RoboDK station: New Station 2.0.1..rdk

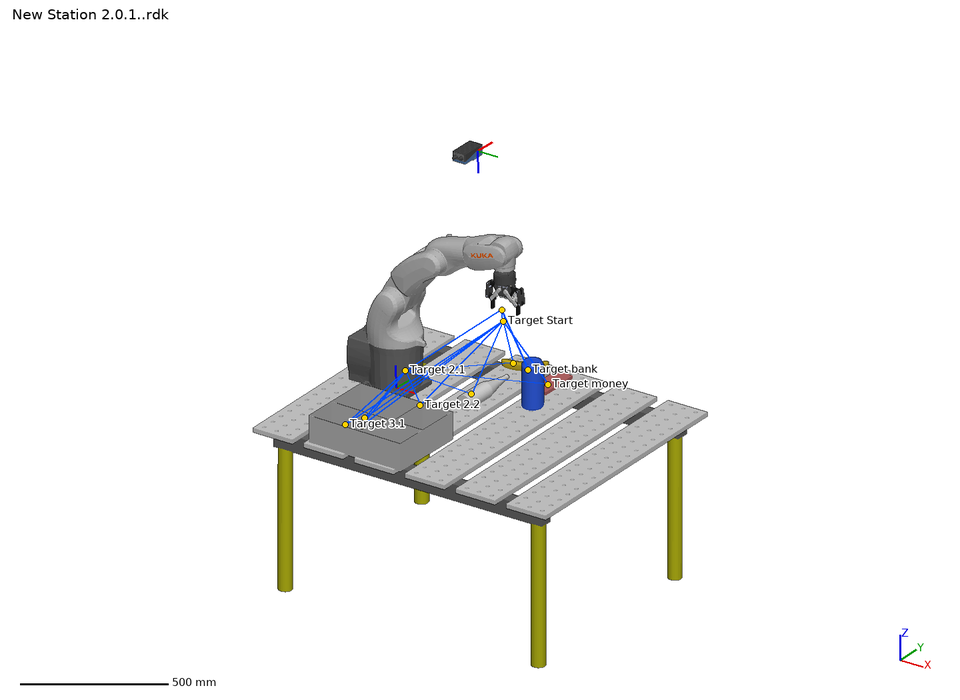
[picture v0: the station drawn from its stored meshes, robots at their saved joint values, targets as dots, program paths as lines]
Station New Station (2). Poses are relative to the parent item; angles as X-Y-Z fixed-axis rotations.
Station parameters (name, value as stored): IO_5, 1, CollisionFreePlanner, KUKA KR 3 R540, CollisionFreePlanner-Rob KUKA KR 3 R540
  - frame KUKA KR 3 R540 Base at (-517.33, 1.06, 0.26) mm, rotated rx -0.44 ry -1.04 rz -0.63 deg
    - robot KUKA KR 3 R540: 6 axes, payload 3 kg, reach 541 mm, repeatability 0.02 mm, weight 26 kg
        modified DH rows (alpha deg, a mm, theta deg, d mm): 0, 0, 0, 345; -90, 20, 0, 0; 0, 260, -90, 0; -90, 20, 0, 260; 90, 0, 0, 0; -90, 0, 180, 75
        joint limits [-170, -170, -110, -175, -120, -350] to [170, 50, 155, 175, 120, 350]; home [0, -90, 90, 0, 0, 0]; saved at [-1.677, -47.408, 34.067, 0.03, 102.342, -1.67]
      - tool Gripper RobotiQ 85 Opened, TCP at (0, -20, 130) mm, size 147.4 x 146.8 x 75 mm
      - tool Gripper RobotiQ 85 Closed, TCP at (0, -20, 130) mm, size 134.4 x 157.6 x 75 mm
    - frame Cam 1 Frame at (362.24, -15.63, 980.06) mm, rotated rx -180 ry -0.87 rz 89.94 deg
      - object Cam 1 at (-36.13, -0.26, 0) mm, rotated rx 0 ry 0 rz -0.06 deg, size 53 x 116 x 38 mm, geometry from Cam2D_SICK_VSPP_5F2113.sld
    - target Target Start (Cartesian target) at (452.7, -7.79, 370.63) mm, rotated rx -180 ry 0 rz 180 deg; joints [-1.545, -47.721, 43.682, 0, 94.039, -1.545] of KUKA KR 3 R540
    - target Target 1 (Cartesian target) at (447.72, -7, 410.9) mm, rotated rx -180 ry 1 rz 180 deg; joints [-1.677, -47.408, 34.067, 0.03, 102.342, -1.67] of KUKA KR 3 R540
    - target Target bank (Cartesian target) at (458.07, 126.15, 139.29) mm, rotated rx 180 ry 0 rz -180 deg; joints [-17.695, -27.719, 59.924, 0, 57.795, -17.695] of KUKA KR 3 R540
    - target Target 2.1 (Cartesian target) at (322.58, -390.29, 298.41) mm, rotated rx 180 ry 1 rz 180 deg; joints [49.256, -36.872, 40.75, -0.76, 85.47, 49.311] of KUKA KR 3 R540
    - target Target 2.2 (Cartesian target) at (321.53, -307.67, 139.3) mm, rotated rx -180 ry 0 rz 180 deg; joints [41.819, -37.777, 80.016, 0, 47.761, 41.819] of KUKA KR 3 R540
    - target Target botlle (Cartesian target) at (290.88, 30.87, 41.6) mm, rotated rx -180 ry 0 rz -180 deg; joints [-9.919, -36.305, 116.095, 0, 10.21, -9.919] of KUKA KR 3 R540
    - target Target 3.1 (Cartesian target) at (123.71, -463.28, 74.82) mm, rotated rx 179 ry 0.04 rz 90 deg; joints [73.166, -17.995, 56.227, -1.21, 51.452, -16.082] of KUKA KR 3 R540
    - target Target banana (Cartesian target) at (247.79, 330.18, 29.97) mm, rotated rx 180 ry 0 rz 120.51 deg; joints [-52.092, -20.233, 74.697, 0, 35.536, -111.581] of KUKA KR 3 R540
    - target Target 3.2 (Cartesian target) at (118.04, -362.03, 29.97) mm, rotated rx 180 ry 0 rz 90.7 deg; joints [69.116, -25.994, 89.591, 0, 26.403, -20.184] of KUKA KR 3 R540
    - target Target money (Cartesian target) at (420.97, 289.96, 12.37) mm, rotated rx -180 ry 0 rz -180 deg; joints [-36.364, 9.152, 14.566, 0, 66.282, -36.364] of KUKA KR 3 R540
    - target Target 3.3 (Cartesian target) at (69.76, -280.26, 13.99) mm, rotated rx 180 ry -0.99 rz 88.58 deg; joints [72.493, -29.84, 112.61, -2.251, 8.17, -16.697] of KUKA KR 3 R540
  - program Prog1 (46 instructions, listed below)
  - program Replace objects (1 instructions, listed below)
  - Python program SimulateToolOpen (listed below)
  - Python program SimulateCamera (listed below)
  - program Target1ToTarget2 (2 instructions, listed below)
  - object  at (-133.86, -215.64, 5.64) mm, rotated rx 90 ry 0 rz -90.4 deg, size 304 x 104 x 379 mm, geometry from  v2.stl
  - object Table at (-140.14, -45.85, 5.02) mm, rotated rx 0 ry 0.02 rz 0.64 deg, size 1193.8 x 965.2 x 609.6 mm, geometry from welding_table.sld
  - object bank v1 at (-54.34, 174.14, 1.34) mm, size 76.9 x 76.9 x 170.3 mm, geometry from bank v1.stl
  - object botlle v1 at (-226.47, -16.86, 5.96) mm, rotated rx -90 ry 0 rz 0 deg, size 60 x 60 x 252.8 mm, geometry from botlle v1.stl
  - object banana v1 at (-288.68, 344.87, 0) mm, rotated rx 0 ry 0 rz -150.16 deg, size 159.5 x 33.3 x 40.6 mm, geometry from banana v1.stl
  - object money v2 at (-132.34, 388.08, 7.15) mm, size 69 x 157 x 12 mm, geometry from money v2.stl
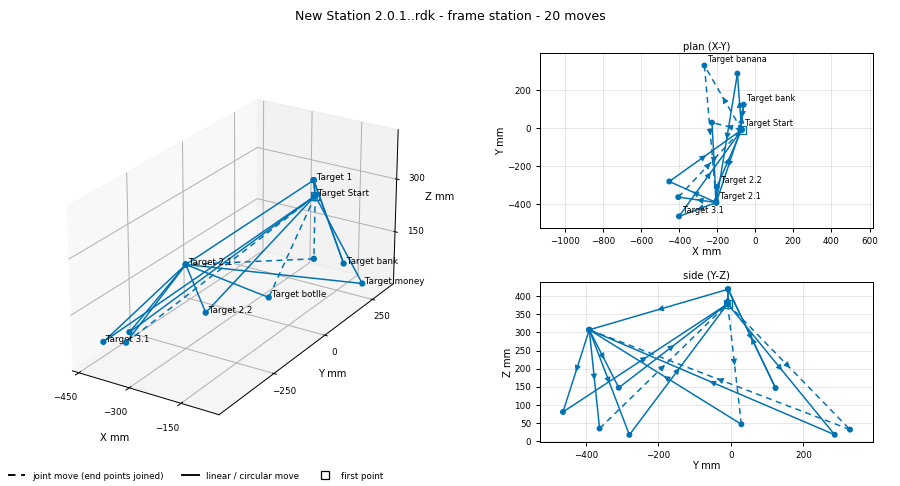
[picture p0: tool path of New Station 2.0.1..rdk in frame station, 20 of 22 moves have a stored position in this frame; points joined in program order, loops and branches not executed]

--- program Prog1 (robot KUKA KR 3 R540) ---
  Set speed (100.0 mm/s)
  Set Tool: Gripper RobotiQ 85 Opened at (0, -20, 130) mm
  Pause 1.5 s
  Call VisibleGripper RobotiQ ...: VisibleGripper RobotiQ 85 Opened_Off
  MoveJ (Target Start)
  MoveL (Target 1)
  MoveL (Target bank)
  Pause 70 ms
  Attach to Gripper RobotiQ 85 Opened
  Pause 50 ms
  MoveL (Target 1)
  MoveL (Target 2.1)
  MoveL (Target 2.2)
  Pause 400 ms
  Detach from Gripper RobotiQ 85 Opened
  Pause 600 ms
  MoveL (Target Start)
  Pause 1.0 s
  MoveJ (Target botlle)
  Attach to Gripper RobotiQ 85 Opened
  Pause 800 ms
  MoveL (Target 2.1)
  MoveL (Target 3.1)
  Detach from Gripper RobotiQ 85 Opened
  Pause 600 ms
  MoveL (Target Start)
  Pause 1.0 s
  MoveJ (Target banana)
  Attach to Gripper RobotiQ 85 Opened
  Pause 600 ms
  MoveJ (Target 2.1)
  MoveL (Target 3.2)
  Detach from Gripper RobotiQ 85 Opened
  Pause 600 ms
  MoveJ (Target Start)
  Pause 1.0 s
  MoveL (Target 10) -> target Target money
  Attach to Gripper RobotiQ 85 Opened
  Pause 600 ms
  MoveL (Target 2.1)
  MoveL (Target 3.3)
  Detach from Gripper RobotiQ 85 Opened
  Pause 600 ms
  MoveL (Target Start)
  MoveL (Target 1)
  Call Replace objects

--- program Replace objects (robot KUKA KR 3 R540) ---
  Replace objects

--- Python program SimulateToolOpen ---
# Type help("robolink") or help("robodk") for more information
# Press F5 to run the script
# Note: you do not need to keep a copy of this file, your python script is saved with the station
from robolink import *    # API to communicate with RoboDK
from robodk import *      # basic matrix operations
RDK = Robolink()

# This file allows simulating the opening and closing of grippers.
# Two models of the gripper per robot are required: one opened and one closed.
# The opened model of the gripper should have the keyword "Opened"
# The closed model of the gripper should have the keyword "Closed"
# Simply place this file in the station and leave it running to
# make it work

OPENED_KEYWORD = 'Opened'
CLOSED_KEYWORD = 'Closed'
UPDATE_FREQUENCY = 0.01

# Loop forever
print('Starting infinite loop to simulate open/close of tools')
while True:
    # First step: get a list of tool pairs (open, closed) per robot
    Tool_Pairs = []
    # get all the robot names (strings)
    all_robots = RDK.ItemList(ITEM_TYPE_ROBOT, True)
    for i in range(len(all_robots)):
        roboti = RDK.Item(all_robots[i])
        roboti_name = roboti.Name()
        # get the tools of each robot
        roboti_tools = roboti.Childs()
        opened = None
        closed = None
        # store the opened model and closed model of each gripper
        for t in range(len(roboti_tools)):
            tnamei = roboti_tools[t].Name()
            if not isinstance(opened,Item) and tnamei.count(OPENED_KEYWORD) > 0:
                opened = roboti_tools[t]
                print('Using %s from robot %s as gripper opened' % (tnamei, roboti_name))
            elif not isinstance(closed,Item) and tnamei.count(CLOSED_KEYWORD) > 0:
                closed = roboti_tools[t]
                print('Using %s from robot %s as gripper closed' % (tnamei, roboti_name))

            if isinstance(opened, Item) and isinstance(closed, Item):
                # Stop if we have an open state and a closed state per robot
                break;
        Tool_Pairs.append([opened, closed])

    # We may find as many pairs of tools as robots are available in the station
    nTool_Pairs = len(Tool_Pairs)
    while True:
        #try:
            # Iterate through all tool pairs and detect the presence of objects
            for i in range(nTool_Pairs):
                opened = Tool_Pairs[i][0]
                closed = Tool_Pairs[i][1]
                open_valid = isinstance(opened,Item)
                close_valid = isinstance(closed,Item)
                tool_is_open = True

                # Check if the tool holds one or more objects:
                if (open_valid and len(opened.Childs()) > 0) or (close_valid and len(closed.Childs()) > 0):
                    tool_is_open = False

                # Update the visibility of the tools
                if open_valid:
                    opened.setVisible(tool_is_open)
                if close_valid:
                    closed.setVisible(not tool_is_open)

            # Take a pause...
            pause(UPDATE_FREQUENCY)

        #except:
            #print('An item was deleted. Remaking tool list')
            #break

--- Python program SimulateCamera ---
# Type help("robolink") or help("robodk") for more information
# Press F5 to run the script
# Documentation: https://robodk.com/doc/en/RoboDK-API.html
# Reference:     https://robodk.com/doc/en/PythonAPI/index.html
# Note: It is not required to keep a copy of this file, your python script is saved with the station
from robolink import *    # RoboDK API
from robodk import *      # Robot toolbox
RDK = Robolink()

# Notify user:
print('To edit this program:\nright click on the Python program, then, select "Edit Python script"')

# Program example:
item = RDK.Item('base')
if item.Valid():
    print('Item selected: ' + item.Name())
    print('Item posistion: ' + repr(item.Pose()))

print('Items in the station:')
itemlist = RDK.ItemList()
print(itemlist)

raise Exception('Program not edited.')

--- program Target1ToTarget2 (robot KUKA KR 3 R540) ---
  MoveJ (Pt 1 (S1)) to (467.86, -0.09, 338.09) mm, rotated rx 179.55 ry -0.28 rz -179.37 deg; joints [-2.236, -43.368, 43.433, -0.46, 90.207, -1.607]
  MoveJ (Pt 2 (S2)) to (745, -20, 365) mm, rotated rx 0 ry 90 rz 0 deg; joints [0, 0, 0, 0, 0, 0]
